INTERFACE I_InputPortChangedEvent EXTENDS I_Event

PROPERTY PUBLIC Target : I_InputPort
GET
END_GET
END_PROPERTY

END_INTERFACE

(* stored: Version 1.1.0.1, ProductVersion 3.1.4024.12
   Itf I_InputPortChangedEvent: Id {fc6b9397-1eec-009e-0f99-fecc75499e00}
   Property Target: Id {76feecca-368f-00fb-3447-79a217ca040e}
   Get Get: Id {f7e5be38-a1d8-0821-3c19-bdcf3b0a69a4} *)
